PROGRAM RETURN_FUKUDA
VAR_INPUT

END_VAR

VAR
	TMR_DELAY: TON;
END_VAR

IF 	INPUT_VAR.TRANSPORT_IDX=0 AND 	INPUT_VAR.STATION_RETURN_IDX=0 AND 	INPUT_VAR.JIG_RETURN_IDX =0 THEN
	INPUT_VAR.TRANSPORT_IDX:=	INPUT_VAR.I_CURRENT_TRANSACTION.TRANSPORT_INDEX;
	INPUT_VAR.STATION_RETURN_IDX:=INPUT_VAR.I_CURRENT_TRANSACTION.STATION_NUMBER_RETURN;
	INPUT_VAR.JIG_RETURN_IDX :=	INPUT_VAR.I_CURRENT_TRANSACTION.JIG_INDEX_RETURN;
ELSE
CASE INPUT_VAR.I_CASE OF
0: //standby near lotbox
	IF INPUT_VAR.ACTIVE_ID=6 THEN
		INPUT_VAR.ACTIVE_ID:=1;
	END_IF
	
	INPUT_VAR.TRANSPORT_IDX:=	INPUT_VAR.I_CURRENT_TRANSACTION.TRANSPORT_INDEX;
	INPUT_VAR.STATION_RETURN_IDX:=INPUT_VAR.I_CURRENT_TRANSACTION.STATION_NUMBER_RETURN;
	INPUT_VAR.JIG_RETURN_IDX :=	INPUT_VAR.I_CURRENT_TRANSACTION.JIG_INDEX_RETURN;

	CASE INPUT_VAR.TRANSPORT_IDX OF
		2 : 
			INPUT_VAR.O_STOPPER_TRANSFER_B:=FALSE;			
			FUKUDA_MOVE(STEP_DATA_1:=3,
				STEP_DATA_2:=1,
				STEP_DATA_3:=12,
				STEP_DATA_4:=0,
				STEP_DATA_5:=1);
				INPUT_VAR.O_STOPPER_TRANSFER_B:=FALSE;
		1 : 
			INPUT_VAR.O_STOPPER_TRANSFER_A:=FALSE;
			FUKUDA_MOVE(STEP_DATA_1:=3,
				STEP_DATA_2:=1,
				STEP_DATA_3:=12,
				STEP_DATA_4:=1,
				STEP_DATA_5:=0);
				INPUT_VAR.O_STOPPER_TRANSFER_A:=FALSE;
	END_CASE			
	input_var.O_VACUUM_On:=FALSE;
	input_var.O_VACUUM_OFF:=FALSE;	
	TMR_DELAY(IN:=FALSE);

1://ready for picking up
	IF INPUT_VAR.ACTIVE_ID=6 THEN
		INPUT_VAR.ACTIVE_ID:=1;
	END_IF

		CASE INPUT_VAR.TRANSPORT_IDX OF
		1:
			INPUT_VAR.I_RETURN_DONE_A:=FALSE;
		
		2:
			INPUT_VAR.I_RETURN_DONE_B:=FALSE;
	END_CASE
	FUKUDA_MOVE(STEP_DATA_1:=3,
				STEP_DATA_2:=1,
				STEP_DATA_3:=13,
				STEP_DATA_4:=0,
				STEP_DATA_5:=0);	
			
2://ready for picking up
	IF INPUT_VAR.ACTIVE_ID=6 THEN
		INPUT_VAR.ACTIVE_ID:=1;
	END_IF

	CASE INPUT_VAR.TRANSPORT_IDX OF
	1:		
		IF INPUT_VAR.I_FUKUDA_TRANSFER_AT_BACK_A THEN
		FUKUDA_MOVE(STEP_DATA_1:=INPUT_VAR.TRANSPORT_IDX+4,
				STEP_DATA_2:=1,
				STEP_DATA_3:=11,
				STEP_DATA_4:=0,
				STEP_DATA_5:=0);
		END_IF
	2:
		IF INPUT_VAR.I_FUKUDA_TRANSFER_AT_BACK_B THEN
		FUKUDA_MOVE(STEP_DATA_1:=INPUT_VAR.TRANSPORT_IDX+4,
				STEP_DATA_2:=1,
				STEP_DATA_3:=11,
				STEP_DATA_4:=0,
				STEP_DATA_5:=0);
	END_IF
	END_CASE
	
		
3://placing onto fukuda transport
	IF INPUT_VAR.ACTIVE_ID=6 THEN
		INPUT_VAR.ACTIVE_ID:=1;
	END_IF

	FUKUDA_MOVE(STEP_DATA_1:=INPUT_VAR.TRANSPORT_IDX+4,
				STEP_DATA_2:=2,
				STEP_DATA_3:=11,
				STEP_DATA_4:=0,
				STEP_DATA_5:=0);
	
4://ready for picking up
	IF INPUT_VAR.ACTIVE_ID=6 THEN
		INPUT_VAR.ACTIVE_ID:=1;
	END_IF
	
	FUKUDA_MOVE(STEP_DATA_1:=INPUT_VAR.TRANSPORT_IDX+4,
				STEP_DATA_2:=6,
				STEP_DATA_3:=11,
				STEP_DATA_4:=0,
				STEP_DATA_5:=0);

5://gripping position
	IF INPUT_VAR.ACTIVE_ID=6 THEN
		INPUT_VAR.ACTIVE_ID:=1;
	END_IF
	
	IF NOT input_var.I_VACUUM_On THEN
		FUKUDA_MOVE(STEP_DATA_1:=INPUT_VAR.TRANSPORT_IDX+4,
				STEP_DATA_2:=2,
				STEP_DATA_3:=12,
				STEP_DATA_4:=0,
				STEP_DATA_5:=0);
	ELSE
		input_var.O_VACUUM_On:=TRUE;
		input_var.O_VACUUM_OFF:=FALSE;
	END_IF
	
				
6://vacuum position 
	IF INPUT_VAR.ACTIVE_ID=6 THEN
		INPUT_VAR.ACTIVE_ID:=1;
	END_IF
	
	FUKUDA_MOVE(STEP_DATA_1:=INPUT_VAR.STATION_RETURN_IDX,
				STEP_DATA_2:=3,
				STEP_DATA_3:=INPUT_VAR.JIG_RETURN_IDX,
				STEP_DATA_4:=0,
				STEP_DATA_5:=0);
				
7://vacuum position 
	IF INPUT_VAR.ACTIVE_ID=6 THEN
		INPUT_VAR.ACTIVE_ID:=1;
	END_IF
	TMR_DELAY(IN:=TRUE,PT:=T#1S);
	IF TMR_DELAY.Q THEN
			FUKUDA_MOVE(STEP_DATA_1:=INPUT_VAR.STATION_RETURN_IDX,
				STEP_DATA_2:=3,
				STEP_DATA_3:=14,
				STEP_DATA_4:=0,
				STEP_DATA_5:=0);
	END_IF
				
8://vacuum position 
	IF INPUT_VAR.ACTIVE_ID=6 THEN
		INPUT_VAR.ACTIVE_ID:=1;
	END_IF
	TMR_DELAY(IN:=FALSE);
	FUKUDA_MOVE(STEP_DATA_1:=INPUT_VAR.STATION_RETURN_IDX,
				STEP_DATA_2:=7,
				STEP_DATA_3:=16,
				STEP_DATA_4:=0,
				STEP_DATA_5:=0);
				
9://vacuum position 
	IF INPUT_VAR.ACTIVE_ID=6 THEN
		INPUT_VAR.ACTIVE_ID:=1;
	END_IF
	
	FUKUDA_MOVE(STEP_DATA_1:=INPUT_VAR.STATION_RETURN_IDX,
				STEP_DATA_2:=8,
				STEP_DATA_3:=INPUT_VAR.JIG_RETURN_IDX,
				STEP_DATA_4:=0,
				STEP_DATA_5:=0);
10: //standby near lotbox
	
	IF INPUT_VAR.ACTIVE_ID=6 THEN
		INPUT_VAR.ACTIVE_ID:=1;
	END_IF

	IF input_var.I_VACUUM_ON THEN
		FUKUDA_MOVE(STEP_DATA_1:=INPUT_VAR.STATION_RETURN_IDX,
				STEP_DATA_2:=4,
				STEP_DATA_3:=INPUT_VAR.JIG_RETURN_IDX,
				STEP_DATA_4:=0,
				STEP_DATA_5:=0);
	ELSE
		input_var.O_VACUUM_ON:=FALSE;
		input_var.O_VACUUM_OFF:=TRUE;			
	END_IF
	
				
11://vacuum position 
	IF INPUT_VAR.ACTIVE_ID=6 THEN
		INPUT_VAR.ACTIVE_ID:=1;
	END_IF
	FUKUDA_MOVE(STEP_DATA_1:=INPUT_VAR.STATION_RETURN_IDX,
				STEP_DATA_2:=1,
				STEP_DATA_3:=INPUT_VAR.JIG_RETURN_IDX,
				STEP_DATA_4:=0,
				STEP_DATA_5:=0);
	IF INPUT_VAR.ACTIVE_ID=3 THEN
		input_var.O_VACUUM_ON:=FALSE;
		input_var.O_VACUUM_OFF:=FALSE;	
	END_IF
	
12://vacuum position 
	IF INPUT_VAR.ACTIVE_ID=6 THEN
		INPUT_VAR.ACTIVE_ID:=1;
	END_IF
	FUKUDA_MOVE(STEP_DATA_1:=0,
				STEP_DATA_2:=1,
				STEP_DATA_3:=4,
				STEP_DATA_4:=0,
				STEP_DATA_5:=0);				
		
100:
	
	input_var.O_VACUUM_On:=FALSE;
	input_var.O_VACUUM_OFF:=FALSE;
END_CASE 
END_IF
IF INPUT_VAR.I_CASE=13 THEN
			CASE INPUT_VAR.TRANSPORT_IDX OF
		1:
			INPUT_VAR.I_RETURN_DONE_A:=TRUE;
		
		2:
			INPUT_VAR.I_RETURN_DONE_B:=TRUE;
	END_CASE
	IF INPUT_VAR.I_RETURN_DONE_A OR INPUT_VAR.I_RETURN_DONE_B THEN
		FLAG_VAR.ALLOW_EXECUTE_RETURN_FUKUDA:=FALSE;
		INPUT_VAR.I_CASE:=100;
	END_IF
END_IF

END_PROGRAM

(* stored: Version 1.1.0.1, ProductVersion 3.1.4020.12
   POU RETURN_FUKUDA: Id {edc92af1-d1cc-45b1-ae2a-ddcdd88d746c}, SpecialFunc None *)
